FUNCTION_BLOCK DigitalOutput EXTENDS Automation.OutputDevice<0>
VAR_OUTPUT
	ContactType : CONTACT_TYPE;
	SimulatedContactValue : BOOL;
END_VAR
VAR
	_ClassName : STRING := __POUNAME();

	_CurrentValue : BOOL;
	_PreviousValue : BOOL;

	_PhysicalContactValue AT %Q* : BOOL;
END_VAR

{attribute 'monitoring' := 'call'}
PROPERTY FINAL Changed : BOOL
GET
Changed := _CurrentValue <> _PreviousValue;
END_GET
END_PROPERTY

{attribute 'monitoring' := 'call'}
PROPERTY ClassName : STRING
GET
ClassName := _ClassName;
END_GET
END_PROPERTY

METHOD FB_init : BOOL
VAR_INPUT
	(* if TRUE, the retain variables are initialized (warm start / cold start)*)
	bInitRetains	: BOOL;
	(* if TRUE, the instance afterwards gets moved into the copy code (online change)*)
	bInCopyCode	: BOOL;
	parent : ISimulatable;
	contactType : CONTACT_TYPE;
END_VAR
THIS^.ContactType := contactType;
END_METHOD

METHOD PROTECTED OnUpdateOutputsFromState
VAR_IN_OUT CONSTANT
	executionContext : Automation.AUTOMATION_EXECUTION_CONTEXT;
END_VAR
IF NOT SimulationMode THEN
	_PhysicalContactValue := _CurrentValue;
ELSE
	SimulatedContactValue := _CurrentValue;
END_IF
END_METHOD

{attribute 'monitoring' := 'call'}
PROPERTY Size : ULINT
GET
Size := XSIZEOF(THIS^);
END_GET
END_PROPERTY

{attribute 'monitoring' := 'call'}
PROPERTY SubDevices : REFERENCE TO ARRAY [0.._SubDeviceCount_ - 1] OF IDevice
GET
SubDevices REF= 0;
END_GET
END_PROPERTY

{attribute 'monitoring' := 'call'}
PROPERTY Value : BOOL
GET
Value := _CurrentValue;
END_GET
SET
_PreviousValue := _CurrentValue;
_CurrentValue := Value;
END_SET
END_PROPERTY

END_FUNCTION_BLOCK

(* stored: Version 1.1.0.1
   POU DigitalOutput: Id {00c882bb-0de1-4d65-b6f1-d0df694bfb3e}, SpecialFunc None
   Property Changed: Id {01a5c812-7bcb-40ee-beb8-2111d2bff10d}
   Get Get: Id {7952ae7e-1e32-4e21-ad02-a2b5baf571ff}
   Property ClassName: Id {004ebedb-8d25-4b94-8fe1-e87a1a80e0da}
   Get Get: Id {3febd567-6452-4bd9-9ba7-e16e305a0d7e}
   Method FB_init: Id {0252e830-6aea-4041-8c99-7cd115603daf}
   Method OnUpdateOutputsFromState: Id {85bb5f79-d992-4624-a97a-f74e005eabf2}
   Property Size: Id {20147cd8-4f58-4ec8-9bf2-efdcff01c0dd}
   Get Get: Id {c04cfb17-d8e5-4f71-829a-687ff94f2753}
   Property SubDevices: Id {13f8888f-ee1b-4ceb-815c-a7d9dca347ab}
   Get Get: Id {6a1723e4-eaea-40e0-a4af-917942665786}
   Property Value: Id {848b14c8-ff4e-42f1-84d0-4c9130ca5b8f}
   Get Get: Id {998ae415-763f-4db8-a772-d3ac3df5c5a0}
   Set Set: Id {19530f80-5a6f-4524-910d-5a6d49063051} *)
